{attribute addProperty BoxType "AX5192-0000-0210-0210"}
{attribute addProperty Id "AT_xAT %I*AT_x_15FCA3A680100MDTAT %Q*MDT_C2B17B7F4860WcStateAT %I*WcState_98A4DF7520.250InfoDataAT %I*InfoData_AEB17F4D152190"}
{attribute addProperty CRC "2773434183"}
{attribute addProperty SizeInBites "282"}
{attribute addProperty SizeInBytes "35.25"}
TYPE AX5192_3FB01CDA :
STRUCT
	{attribute addProperty Name "AT_x"}
	AT_x : AT_x_15FCA3A6;
	{attribute addProperty Name "MDT"}
	MDT : MDT_C2B17B7F;
	{attribute addProperty Name "WcState"}
	WcState : WcState_98A4DF75;
	{attribute addProperty Name "InfoData"}
	InfoData : InfoData_AEB17F4D;
END_STRUCT
END_TYPE

(* stored: Version 1.2.0.0, ProductVersion 3.1.4024.9
   DUT AX5192_3FB01CDA: Id {1afd1740-2c4e-47d6-b943-316283797767} *)
